FUNCTION TFCylinder_ClearAllCommand : bool
VAR_INPUT
Command : pointer to  CylinderCommand;
END_VAR
VAR
END_VAR

Command^.ErrorReset := FALSE;
Command^.Deactivation:=FALSE;
Command^.Activation:=FALSE;
Command^.Hold:=FALSE;
Command^.Abort:=FALSE;
Command^.Stop:= FALSE;
TFCylinder_ClearAllCommand:=TRUE;

END_FUNCTION

(* stored: Version 1.1.0.1, ProductVersion 3.1.4024.11
   POU TFCylinder_ClearAllCommand: Id {32ff928a-ad1e-4cd5-8287-0164b59e96b1}, SpecialFunc None *)
